// TIA Portal V20 export
DATA_BLOCK "LPFE_FromHostBuffer"   // DB247
TITLE = FromHostBuffer
// Contains Interface channel components for FromHost channel
// stored: Access Published, DBAccessibleFromWebserver false, MemoryReserve 100, Namespace PFE
   VAR
      inChannel { ExternalVisible := 'False'} : "LPFE_typePFEDataInChannel";   // Channel for inbound messages
   END_VAR
BEGIN
   // inChannel.msgFromKepserver : Array of DINT used for direct tag communication from Kepserver
END_DATA_BLOCK
